// TIA Portal V21 export
FUNCTION_BLOCK "AUX MES"   // FB1000, LAD
{ S7_Optimized_Access := 'FALSE' }
// stored: AutoNumber false, SetENOAutomatically false
   VAR
      DATI { S7_SetPoint := 'True'} : "UDT_MES";
      TOUT { S7_SetPoint := 'True'} : IEC_TIMER;
      FP1 : Bool;
      FP2 : Bool;
      COMM_ERROR : Bool;
      IndexPID : Int;
      AllarmePresenteSterilizzatore { ExternalVisible := 'False'; ExternalWritable := 'False'} : Bool;
      AllarmePresentePID : Bool;
   END_VAR
   VAR_TEMP
      LIFE_IMP : Bool;
      ON : Bool;
      RIPORTO : Bool;
      RICETTA_DIVERSA : Bool;
      RICHIESTA_CAMBIO_RICETTA : Bool;
      "Counter" : Int;
      AppoAllarme : Bool;
   END_VAR
   VAR_TEMP   // added for the SCL form of the ladder/FBD networks
      _w1 : Bool;
      _w2 : Bool;
   END_VAR
BEGIN

REGION Network 1: on bit
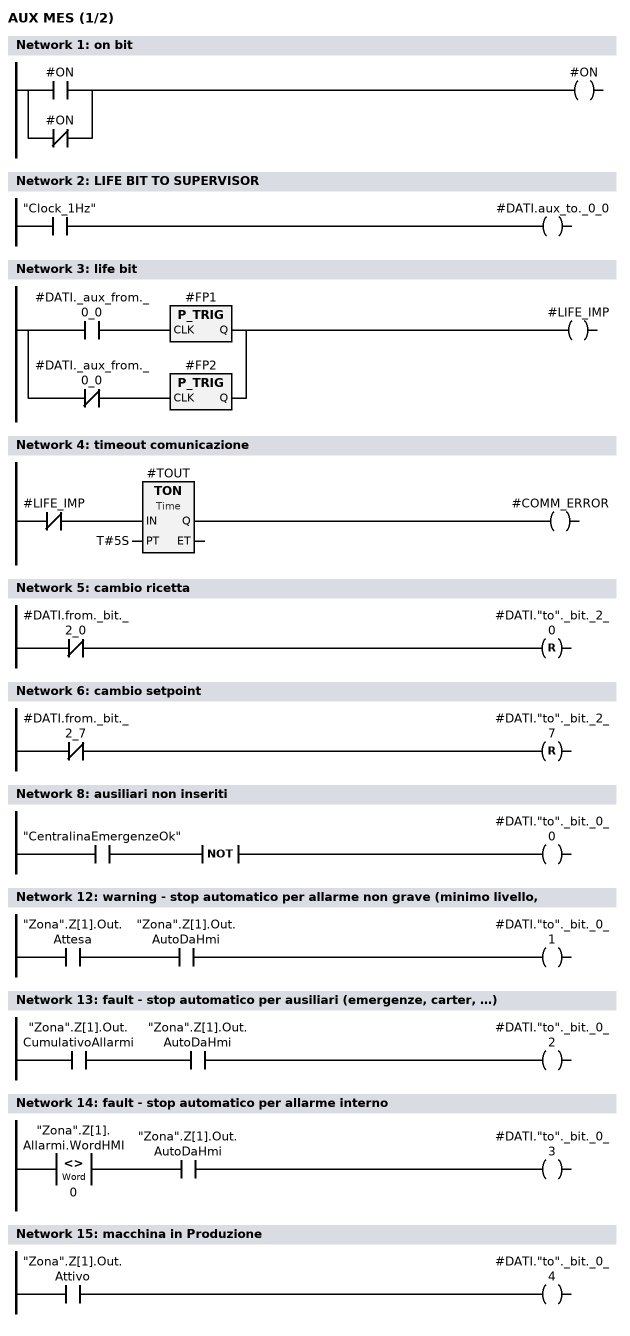
   RUNG wire#powerrail
      Contact( #ON )
      wire#w1
      Coil( #ON )
   END_RUNG
   RUNG wire#powerrail
      I_Contact( #ON )
   END_RUNG wire#w1
   // the same network as SCL:
   #ON := #ON OR NOT #ON;
END_REGION

REGION Network 2: LIFE BIT TO SUPERVISOR
   RUNG wire#powerrail
      Contact( "Clock_1Hz" )
      Coil( #DATI.aux_to._0_0 )
   END_RUNG
   // the same network as SCL:
   #DATI.aux_to._0_0 := "Clock_1Hz";
END_REGION

REGION Network 3: life bit
   RUNG wire#powerrail
      Contact( #DATI._aux_from._0_0 )
      P_Trig( #FP1 )
      wire#w1
      Coil( #LIFE_IMP )
   END_RUNG
   RUNG wire#powerrail
      I_Contact( #DATI._aux_from._0_0 )
      P_Trig( #FP2 )
   END_RUNG wire#w1
   // the same network as SCL:
   #_w1 := #DATI._aux_from._0_0 AND NOT #FP1;   // rising edge
   #FP1 := #DATI._aux_from._0_0;
   #_w2 := NOT #DATI._aux_from._0_0 AND NOT #FP2;   // rising edge
   #FP2 := NOT #DATI._aux_from._0_0;
   #LIFE_IMP := #_w1 OR #_w2;
END_REGION

REGION Network 4: timeout comunicazione
   RUNG wire#powerrail
      I_Contact( #LIFE_IMP )
      { S7_Templates := "time_type := Time" } #TOUT.TON(pt := T#5S, et =>)
      Coil( #COMM_ERROR )
   END_RUNG
   // the same network as SCL:
   #TOUT.TON(IN := NOT #LIFE_IMP, PT := T#5S);
   #COMM_ERROR := #TOUT.Q;
END_REGION

REGION Network 5: cambio ricetta
   RUNG wire#powerrail
      I_Contact( #DATI.from._bit._2_0 )
      R_Coil( #DATI."to"._bit._2_0 )
   END_RUNG
   // the same network as SCL:
   IF NOT #DATI.from._bit._2_0 THEN #DATI."to"._bit._2_0 := FALSE; END_IF;
END_REGION

REGION Network 6: cambio setpoint
   RUNG wire#powerrail
      I_Contact( #DATI.from._bit._2_7 )
      R_Coil( #DATI."to"._bit._2_7 )
   END_RUNG
   // the same network as SCL:
   IF NOT #DATI.from._bit._2_7 THEN #DATI."to"._bit._2_7 := FALSE; END_IF;
END_REGION

REGION Network 7 (SCL): Valori analogici
   #DATI.to._dint._0_06 := "Analogica".A[K_Analogica_LivelloVascaProdotto].Out.AnalogicaAttuale.Valore;
   #DATI.to._dint._0_09 := "Analogica".A[K_Analogica_TemperaturaUscitaSterilizzatoreProcesso].Out.AnalogicaAttuale.Valore;
   #DATI.to._dint._0_010 := "Analogica".A[K_Analogica_TemperaturaUscitaSosta].Out.AnalogicaAttuale.Valore;
   #DATI.to._dint._0_011 := "Analogica".A[K_Analogica_TemperaturaUscitaRaffredatoreProcesso].Out.AnalogicaAttuale.Valore;
   #DATI.to._dint._0_012 := "Analogica".A[K_Analogica_PortataIngressoProdotto].Out.AnalogicaAttuale.Valore;
   #DATI.to._dint._0_013 := "Analogica".A[K_Analogica_PressioneSicurezzaIngressoSterilizzatore].Out.AnalogicaAttuale.Valore;
END_REGION

REGION Network 8: ausiliari non inseriti
   RUNG wire#powerrail
      Contact( "CentralinaEmergenzeOk" )
      Not()
      Coil( #DATI."to"._bit._0_0 )
   END_RUNG
   // the same network as SCL:
   #DATI."to"._bit._0_0 := NOT "CentralinaEmergenzeOk";
END_REGION

REGION Network 9 (SCL): Allarmi strumenti sterilizzatore
   // #AppoAllarme := FALSE;
   // FOR #Counter := 0 TO 20 DO
   //     IF "Analogica".A[#Counter].Allarmi.WordHMI <> 0 THEN
   //         #AppoAllarme := TRUE;
   //     END_IF;
   // END_FOR;

   // #AllarmePresenteSterilizzatore := #AppoAllarme;
END_REGION

REGION Network 10 (SCL): Verifico allarmi PID
   // #AppoAllarme := FALSE;
   // FOR #Counter := 0 TO 20 DO
   //     IF "Pid".P[#Counter].Allarmi.A[1].Stato  OR
   //         "Pid".P[#Counter].Allarmi.A[2].Stato OR
   //         "Pid".P[#Counter].Allarmi.A[3].Stato THEN
   //         #AppoAllarme := TRUE;
   //     END_IF;
   // END_FOR;

   // #AllarmePresentePID := #AppoAllarme;
END_REGION

NETWORK
TITLE = allarme PID
//      L     #IndexPID
//      L     30
//      <=I
//      JC    Q201_1

//      L     0
//      T     #IndexPID
//      CLR
//      =     #AllarmePresentePID

//Q201_1 : NOP 0

REGION Network 12: warning - stop automatico per allarme non grave (minimo livello,
   RUNG wire#powerrail
      Contact( "Zona".Z[1].Out.Attesa )
      Contact( "Zona".Z[1].Out.AutoDaHmi )
      Coil( #DATI."to"._bit._0_1 )
   END_RUNG
   // the same network as SCL:
   #DATI."to"._bit._0_1 := "Zona".Z[1].Out.Attesa AND "Zona".Z[1].Out.AutoDaHmi;
END_REGION

REGION Network 13: fault - stop automatico per ausiliari (emergenze, carter, …)
   RUNG wire#powerrail
      Contact( "Zona".Z[1].Out.CumulativoAllarmi )
      Contact( "Zona".Z[1].Out.AutoDaHmi )
      Coil( #DATI."to"._bit._0_2 )
   END_RUNG
   // the same network as SCL:
   #DATI."to"._bit._0_2 := "Zona".Z[1].Out.CumulativoAllarmi AND "Zona".Z[1].Out.AutoDaHmi;
END_REGION

REGION Network 14: fault - stop automatico per allarme interno
   RUNG wire#powerrail
      { S7_Templates := "SrcType := Word" } NE_Contact(in1 := "Zona".Z[1].Allarmi.WordHMI, in2 := 0)
      Contact( "Zona".Z[1].Out.AutoDaHmi )
      Coil( #DATI."to"._bit._0_3 )
   END_RUNG
   // the same network as SCL:
   #DATI."to"._bit._0_3 := ("Zona".Z[1].Allarmi.WordHMI <> 0) AND "Zona".Z[1].Out.AutoDaHmi;
END_REGION

REGION Network 15: macchina in Produzione
   RUNG wire#powerrail
      Contact( "Zona".Z[1].Out.Attivo )
      Coil( #DATI."to"._bit._0_4 )
   END_RUNG
   // the same network as SCL:
   #DATI."to"._bit._0_4 := "Zona".Z[1].Out.Attivo;
END_REGION

REGION Network 16 (SCL): NomeRicetta Mes
   //#DATI.from._string._0_00:="MacchinaARicetta".M[1].Archivio[#DATI.from._dint._0_00].NomeFormato;
   #DATI.to._dint._0_00 := "MacchinaARicetta".M[1].Hmi.Indice_RicettaAttuale;
   #DATI.to._string._0_00 := "MacchinaARicetta".M[1].Lavoro.NomeFormato;
END_REGION

REGION Network 17 (SCL): Bit Pompa Mono
   #DATI.to._bit._0_5 := "MacchinaARicetta".M[1].Lavoro.DatoBool[1];
END_REGION

REGION Network 18: RICETTA DIVERSA
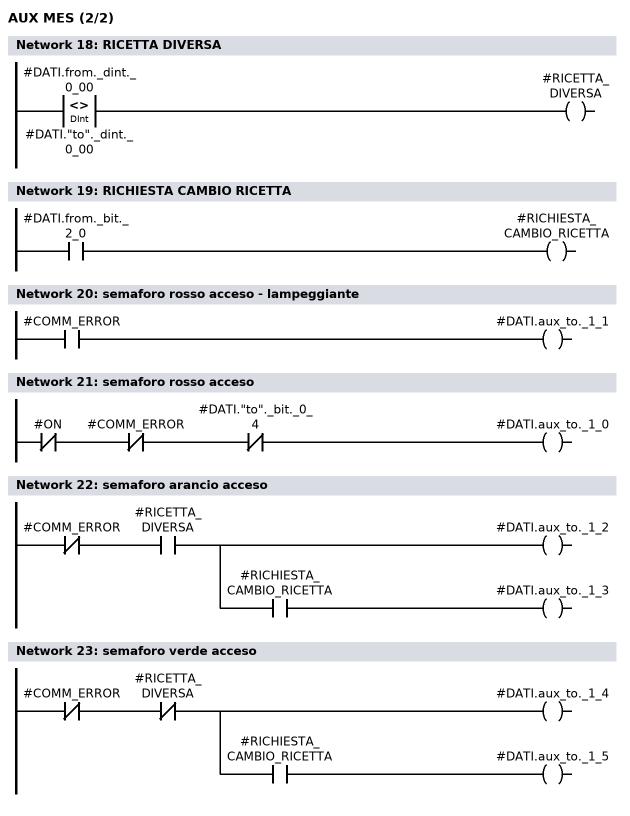
   RUNG wire#powerrail
      { S7_Templates := "SrcType := DInt" } NE_Contact(in1 := #DATI.from._dint._0_00, in2 := #DATI."to"._dint._0_00)
      Coil( #RICETTA_DIVERSA )
   END_RUNG
   // the same network as SCL:
   #RICETTA_DIVERSA := #DATI.from._dint._0_00 <> #DATI."to"._dint._0_00;
END_REGION

REGION Network 19: RICHIESTA CAMBIO RICETTA
   RUNG wire#powerrail
      Contact( #DATI.from._bit._2_0 )
      Coil( #RICHIESTA_CAMBIO_RICETTA )
   END_RUNG
   // the same network as SCL:
   #RICHIESTA_CAMBIO_RICETTA := #DATI.from._bit._2_0;
END_REGION

REGION Network 20: semaforo rosso acceso - lampeggiante
   RUNG wire#powerrail
      Contact( #COMM_ERROR )
      Coil( #DATI.aux_to._1_1 )
   END_RUNG
   // the same network as SCL:
   #DATI.aux_to._1_1 := #COMM_ERROR;
END_REGION

REGION Network 21: semaforo rosso acceso
   RUNG wire#powerrail
      I_Contact( #ON )
      I_Contact( #COMM_ERROR )
      I_Contact( #DATI."to"._bit._0_4 )
      Coil( #DATI.aux_to._1_0 )
   END_RUNG
   // the same network as SCL:
   #DATI.aux_to._1_0 := NOT #ON AND NOT #COMM_ERROR AND NOT #DATI."to"._bit._0_4;
END_REGION

REGION Network 22: semaforo arancio acceso
   RUNG wire#powerrail
      I_Contact( #COMM_ERROR )
      Contact( #RICETTA_DIVERSA )
      wire#w1
      Coil( #DATI.aux_to._1_2 )
   END_RUNG
   RUNG wire#w1
      Contact( #RICHIESTA_CAMBIO_RICETTA )
      Coil( #DATI.aux_to._1_3 )
   END_RUNG
   // the same network as SCL:
   #DATI.aux_to._1_2 := NOT #COMM_ERROR AND #RICETTA_DIVERSA;
   #DATI.aux_to._1_3 := #DATI.aux_to._1_2 AND #RICHIESTA_CAMBIO_RICETTA;
END_REGION

REGION Network 23: semaforo verde acceso
   RUNG wire#powerrail
      I_Contact( #COMM_ERROR )
      I_Contact( #RICETTA_DIVERSA )
      wire#w1
      Coil( #DATI.aux_to._1_4 )
   END_RUNG
   RUNG wire#w1
      Contact( #RICHIESTA_CAMBIO_RICETTA )
      Coil( #DATI.aux_to._1_5 )
   END_RUNG
   // the same network as SCL:
   #DATI.aux_to._1_4 := NOT #COMM_ERROR AND NOT #RICETTA_DIVERSA;
   #DATI.aux_to._1_5 := #DATI.aux_to._1_4 AND #RICHIESTA_CAMBIO_RICETTA;
END_REGION
END_FUNCTION_BLOCK
